% RSLogix 500 project PLC1_FINALPROJECT.RSS, saved by version 12.00.00.00 %
PROJECT "UNTITLED"    % processor: Bul.1763 MicroLogix 1100 Series B %

PROGRAM FILES
  LAD 2   9 rungs

DATA FILES
  O0 OUTPUT  5 elements
  I1 INPUT  6 elements
  S2 STATUS  66 elements
  B3 BINARY  1 elements
  T4 TIMER  5 elements
  C5 COUNTER  10 elements
  R6 CONTROL  1 elements
  N7 INTEGER  1 elements
  F8 FLOAT  5 elements

LADDER 2
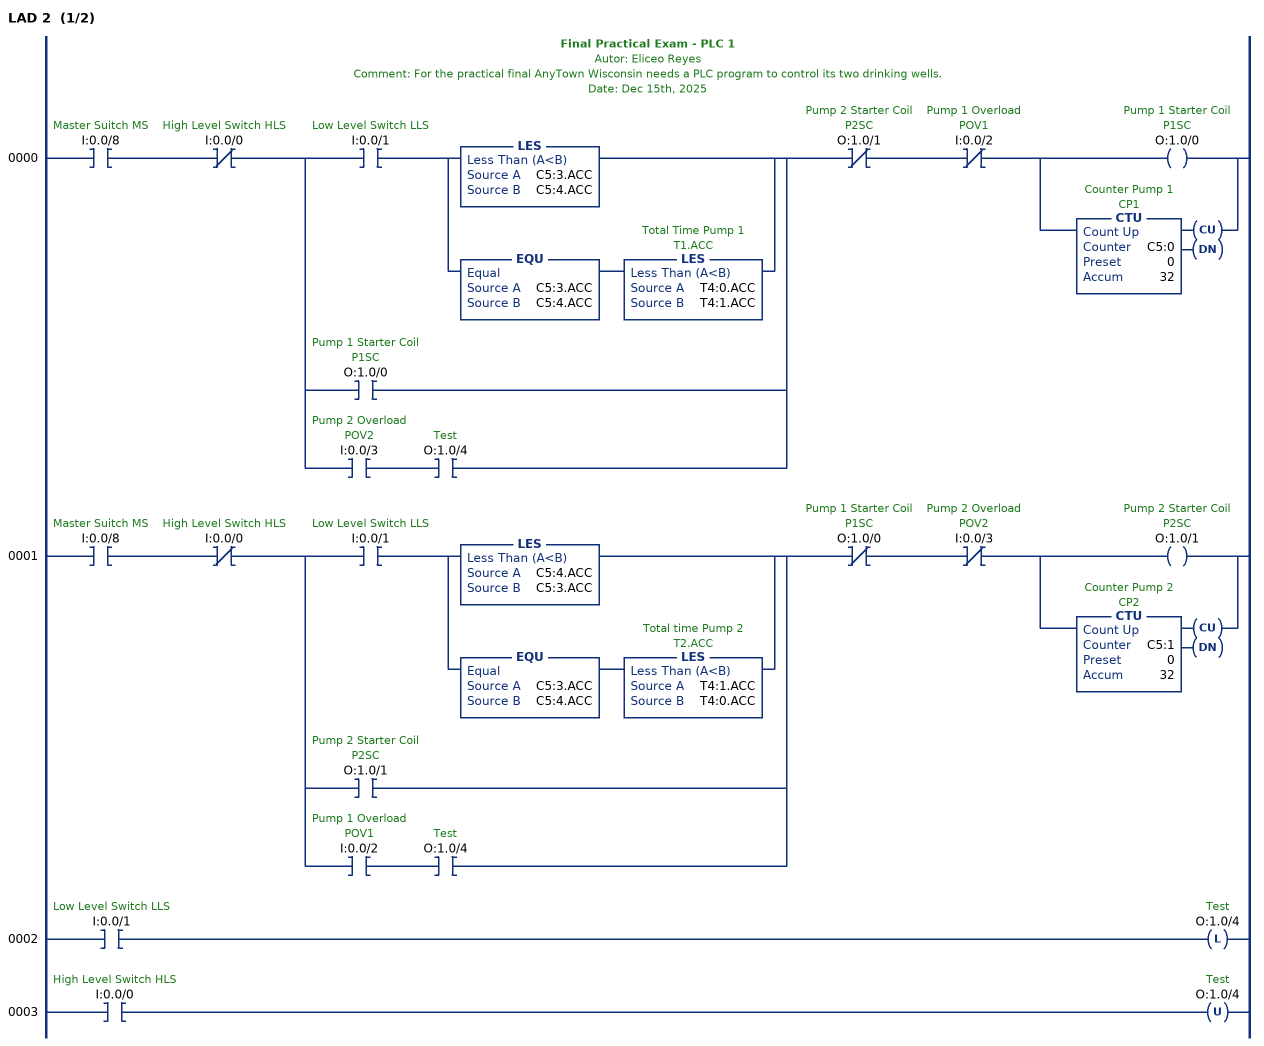
% Rung: 0 %
% TITLE: Final Practical Exam - PLC 1 %
% Autor: Eliceo Reyes
% Comment: For the practical final AnyTown Wisconsin needs a PLC program to control its two drinking wells.
% Date: Dec 15th, 2025 %
SOR XIC I:0.0/8 XIO I:0.0/0 BST XIC I:0.0/1 BST LES C5:3.ACC C5:4.ACC NXB EQU C5:3.ACC C5:4.ACC LES T4:0.ACC T4:1.ACC BND NXB XIC O:1.0/0 NXB XIC I:0.0/3 XIC O:1.0/4 BND XIO O:1.0/1 XIO I:0.0/2 BST OTE O:1.0/0 NXB CTU C5:0 0 32 BND EOR
%   I:0.0/8  MS  "Master Suitch" %
%   I:0.0/0  HLS  "High Level Switch" %
%   I:0.0/1  LLS  "Low Level Switch" %
%   T4:0  T1  "Total Time Pump 1" %
%   T4:1  T2  "Total time Pump 2" %
%   O:1.0/0  P1SC  "Pump 1 Starter Coil" %
%   I:0.0/3  POV2  "Pump 2 Overload" %
%   O:1.0/4  "Test" %
%   O:1.0/1  P2SC  "Pump 2 Starter Coil" %
%   I:0.0/2  POV1  "Pump 1 Overload" %
%   C5:0  CP1  "Counter Pump 1" %
% Rung: 1 %
SOR XIC I:0.0/8 XIO I:0.0/0 BST XIC I:0.0/1 BST LES C5:4.ACC C5:3.ACC NXB EQU C5:3.ACC C5:4.ACC LES T4:1.ACC T4:0.ACC BND NXB XIC O:1.0/1 NXB XIC I:0.0/2 XIC O:1.0/4 BND XIO O:1.0/0 XIO I:0.0/3 BST OTE O:1.0/1 NXB CTU C5:1 0 32 BND EOR
%   I:0.0/8  MS  "Master Suitch" %
%   I:0.0/0  HLS  "High Level Switch" %
%   I:0.0/1  LLS  "Low Level Switch" %
%   T4:1  T2  "Total time Pump 2" %
%   T4:0  T1  "Total Time Pump 1" %
%   O:1.0/1  P2SC  "Pump 2 Starter Coil" %
%   I:0.0/2  POV1  "Pump 1 Overload" %
%   O:1.0/4  "Test" %
%   O:1.0/0  P1SC  "Pump 1 Starter Coil" %
%   I:0.0/3  POV2  "Pump 2 Overload" %
%   C5:1  CP2  "Counter Pump 2" %
% Rung: 2 %
SOR XIC I:0.0/1 OTL O:1.0/4 EOR
%   I:0.0/1  LLS  "Low Level Switch" %
%   O:1.0/4  "Test" %
% Rung: 3 %
SOR XIC I:0.0/0 OTU O:1.0/4 EOR
%   I:0.0/0  HLS  "High Level Switch" %
%   O:1.0/4  "Test" %

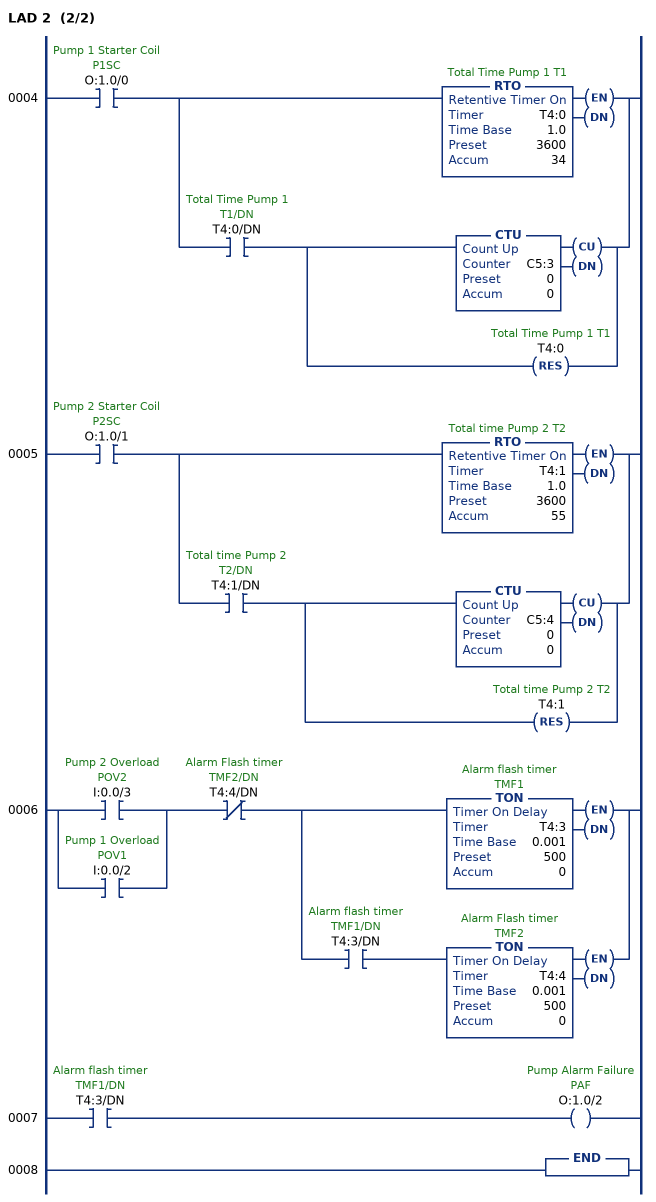
% Rung: 4 %
SOR XIC O:1.0/0 BST RTO T4:0 1.0 3600 34 NXB XIC T4:0/DN BST CTU C5:3 0 0 NXB RES T4:0 BND BND EOR
%   O:1.0/0  P1SC  "Pump 1 Starter Coil" %
%   T4:0  T1  "Total Time Pump 1" %
% Rung: 5 %
SOR XIC O:1.0/1 BST RTO T4:1 1.0 3600 55 NXB XIC T4:1/DN BST CTU C5:4 0 0 NXB RES T4:1 BND BND EOR
%   O:1.0/1  P2SC  "Pump 2 Starter Coil" %
%   T4:1  T2  "Total time Pump 2" %
% Rung: 6 %
SOR BST XIC I:0.0/3 NXB XIC I:0.0/2 BND XIO T4:4/DN BST TON T4:3 0.001 500 0 NXB XIC T4:3/DN TON T4:4 0.001 500 0 BND EOR
%   I:0.0/3  POV2  "Pump 2 Overload" %
%   I:0.0/2  POV1  "Pump 1 Overload" %
%   T4:4  TMF2  "Alarm Flash timer" %
%   T4:3  TMF1  "Alarm flash timer" %
% Rung: 7 %
SOR XIC T4:3/DN OTE O:1.0/2 EOR
%   T4:3  TMF1  "Alarm flash timer" %
%   O:1.0/2  PAF  "Pump Alarm Failure" %
% Rung: 8 %
SOR END EOR

OTHER DOCUMENTED ADDRESSES
  B3:0/0  "Pump station enable"
  C2  "Counter Pump 2"
  O:0.0/1  "Green Light"
  O:1.0/3  "test"
  T  "Timer Pump 1"
  XIO  

COMMENTS NOT ATTACHED TO A CURRENT RUNG
  O:1.0/0: PLC 1 Final Project / Author: Eliceo Reyes
    Comment: Final Project PLC 1
    Date: Dec 15, 2025

DATA TABLE (non-zero values as saved)
DATA T4
% .PRE .ACC %
% T4:0 % 3600 34
% T4:1 % 3600 55
% T4:3 % 500 0
% T4:4 % 500 0
DATA C5
% .PRE .ACC %
% C5:0 % 0 32
% C5:1 % 0 32
DATA F8
% F8:0 % 0 0.004166667 0 0 0
